{attribute 'qualified_only'}
{attribute 'strict'}
{attribute 'to_string'}
TYPE E_FactoryOpMode :
(
    HALTED,
	RUNNING,
    PAUSED,
    RESET
);
END_TYPE

(* stored: Version 1.1.0.1
   DUT E_FactoryOpMode: Id {c316459d-1ae2-4750-830f-f6e7f48ab971} *)
